(* CODESYS project WagoAppKNX.ecp

Project tree, tasks and I/O mapping:
  Steuerung : 750-8202 PFC200 2ETH RS, WAGO, order no. 0750-8202, version 5.14.3.31
    application Firmware_15
      libraries: ; WagoAppKNX, 1.0.2.6 (WAGO); VisuDialogs, * (System)
      task PLC_Task (cyclic, interval t#50ms, priority 15) calls PLC_PRG
      task VISU_TASK (cyclic, interval 100 ms, priority 15) calls VisuElems.Visu_Prg
      program PLC_PRG [CFC]
      visualisation Visualization
      Symbols
      program PLC_PRG_TP [CFC]
      visualisation Visualization_TM
    Kbus : Kbus, WAGO, version 1.4.0.2
        unmapped channels: K-BUS diagnostics
      KNX_EIB_TP1_Interface : 0753-0646, WAGO, order no. 0753-0646, version 0.0.0.10
          settings: K-BUS Module slot index = 1
          unmapped channels: _INPUTCHANNEL, _OUTPUTCHANNEL
    MODBUS
      MODBUS : MODBUS, WAGO, order no. n/a, version 1.1.1.15
    Serial
      COM1 : COM1, WAGO, version 0.0.0.19
  PFC200_2ETH_RS : 750-8202 PFC200 2ETH RS, WAGO, order no. 0750-8202, version 5.14.3.31
    application Application
      libraries: ; WagoAppKNX, 1.0.4.11 (WAGO)
      task PLC_Task (cyclic, interval t#50ms, priority 15) calls PLC_PRG
      program PLC_PRG [CFC]
    Kbus : Kbus, WAGO, version 1.4.0.2
        unmapped channels: K-BUS diagnostics
      _8_DI_Generic : 075x-8DI, WAGO, order no. 075x-8DI, version 0.0.0.13
          unmapped channels: _IN
      _2_DO_Generic : 075x-2DO, WAGO, order no. 075x-2DO, version 0.0.0.13
          unmapped channels: _OUT
      KNX_EIB_TP1_Interface : 0753-0646, WAGO, order no. 0753-0646, version 0.0.0.10
          unmapped channels: _INPUTCHANNEL, _OUTPUTCHANNEL
    MODBUS
      MODBUS : MODBUS, WAGO, order no. n/a, version 1.1.1.15
    Serial
      COM1 : COM1, WAGO, version 0.0.0.19
  PFC200_2ETH_RS_1 : 750-8202 PFC200 2ETH RS, WAGO, order no. 0750-8202, version 5.16.3.16
    application Firmware_19
      libraries: ; WagoAppKNX, 1.0.4.11 (WAGO); WagoSysKbusModule, 1.8.4.4 (WAGO); VisuDialogs, * (System)
      task PLC_Task (cyclic, interval t#50ms, priority 15) calls PLC_PRG
      task VISU_TASK (cyclic, interval 100 ms, priority 15) calls VisuElems.Visu_Prg
      program PLC_PRG [CFC]
      visualisation Visualization
      Symbols
    Kbus : Kbus, WAGO, version 1.4.0.2
        unmapped channels: K-BUS diagnostics
      KNX_EIB_TP1_Interface : 0753-0646, WAGO, order no. 0753-0646, version 0.0.0.10
          settings: K-BUS Module slot index = 1
          unmapped channels: _INPUTCHANNEL, _OUTPUTCHANNEL
    MODBUS
      MODBUS : MODBUS, WAGO, order no. n/a, version 1.1.1.16
    Serial
      COM1 : COM1, WAGO, version 0.0.0.19
  Firmware_11 : 750-8202 PFC200 2ETH RS, WAGO, order no. 0750-8202, version 5.11.1.16
    application Firmware_11
      libraries: ; WagoAppKNX, * (WAGO)
      task PLC_Task (cyclic, interval t#50ms, priority 15) calls PLC_PRG
      task VISU_TASK (cyclic, interval 100 ms, priority 15) calls VisuElems.Visu_Prg
      program PLC_PRG [CFC]
      Symbols
      visualisation Visualization
    Kbus : Kbus, WAGO, version 1.4.0.2
        unmapped channels: K-BUS diagnostics
      _16_DI_Generic : 075x-16DI, WAGO, order no. 075x-16DI, version 0.0.0.13
          settings: K-BUS Module slot index = 1
          unmapped channels: _IN
      _16_DI_Generic_1 : 075x-16DI, WAGO, order no. 075x-16DI, version 0.0.0.13
          settings: K-BUS Module slot index = 2
          unmapped channels: _IN
      _16_DI_Generic_2 : 075x-16DI, WAGO, order no. 075x-16DI, version 0.0.0.13
          settings: K-BUS Module slot index = 3
          unmapped channels: _IN
      _8_DI_Generic : 075x-8DI, WAGO, order no. 075x-8DI, version 0.0.0.13
          settings: K-BUS Module slot index = 4
          unmapped channels: _IN
      _8_DI_Generic_1 : 075x-8DI, WAGO, order no. 075x-8DI, version 0.0.0.13
          settings: K-BUS Module slot index = 5
          unmapped channels: _IN
      _16_DO_Generic : 075x-16DO, WAGO, order no. 075x-16DO, version 0.0.0.13
          settings: K-BUS Module slot index = 6
          unmapped channels: _OUT
      _16_DO_Generic_1 : 075x-16DO, WAGO, order no. 075x-16DO, version 0.0.0.13
          settings: K-BUS Module slot index = 7
          unmapped channels: _OUT
      _16_DO_Generic_2 : 075x-16DO, WAGO, order no. 075x-16DO, version 0.0.0.13
          settings: K-BUS Module slot index = 8
          unmapped channels: _OUT
      KNX_EIB_TP1_Interface : 0753-0646, WAGO, order no. 0753-0646, version 0.0.0.10
          settings: K-BUS Module slot index = 9
          unmapped channels: _INPUTCHANNEL, _OUTPUTCHANNEL
      DALI_MULTI_MASTER_MODULE : 0753-0647, WAGO, order no. 0753-0647, version 0.0.0.20
          settings: K-BUS Module slot index = 10
          unmapped channels: _IN, _OUT
    MODBUS
      MODBUS : MODBUS, WAGO, order no. n/a, version 1.1.1.15
    Serial
      COM1 : COM1, WAGO, version 0.0.0.19
  libraries: VisuSymbols, 4.1.0.0 (System); WagoVisuIcons, 1.1.0.5 (WAGO); WagoVisuIconsMaterialDesign, 1.0.0.0 (WAGO)
  text list GlobalTextList
*)

// Steuerung/Firmware_15/PLC_PRG
PROGRAM PLC_PRG
VAR
	KNX_Master: FbKNX_Master;
	oStatus: WagoAppKNX.WagoSysErrorBase.FbResult;
	sStatus: STRING;
	xProgMode: BOOL;
	wCountFbDPT: WORD;
	M1_001_DPT_Switch_Control: WagoAppKNX.FbDPT_Switch_Control;
	xUpdate_PLC: BOOL;
	xControl_OUT: BOOL;
	xSwitch_OUT: BOOL;
	dwIndex_DPT: DWORD := 1;
	xSwitch_IN: BOOL;
	xControl_IN: BOOL;
	xUpdate_KNX: BOOL;
END_VAR

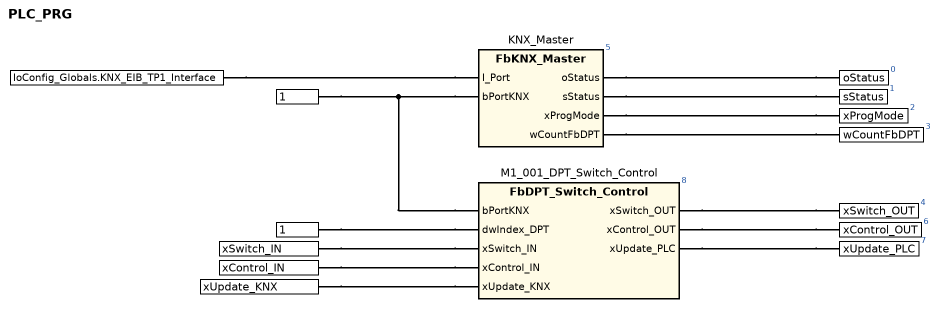
oStatus := KNX_Master.oStatus;
sStatus := KNX_Master.sStatus;
xProgMode := KNX_Master.xProgMode;
wCountFbDPT := KNX_Master.wCountFbDPT;
xSwitch_OUT := M1_001_DPT_Switch_Control.xSwitch_OUT;
KNX_Master(I_Port := IoConfig_Globals.KNX_EIB_TP1_Interface, bPortKNX := 1); // FbKNX_Master
xControl_OUT := M1_001_DPT_Switch_Control.xControl_OUT;
xUpdate_PLC := M1_001_DPT_Switch_Control.xUpdate_PLC;
M1_001_DPT_Switch_Control(
    bPortKNX := 1,
    dwIndex_DPT := 1,
    xSwitch_IN := xSwitch_IN,
    xControl_IN := xControl_IN,
    xUpdate_KNX := xUpdate_KNX); // FbDPT_Switch_Control

END_PROGRAM

// PFC200_2ETH_RS/Application/PLC_PRG
PROGRAM PLC_PRG
VAR
	KNX_Master: FbKNX_Master;
	oStatus: WagoAppKNX.WagoSysErrorBase.FbResult;
	sStatus: STRING;
	xProgMode: BOOL;
	wCountFbDPT: WORD;
	M1_001_DPT_Switch_Control: WagoAppKNX.FbDPT_Switch_Control;
	xUpdate_PLC: BOOL;
	xControl_OUT: BOOL;
	xSwitch_OUT: BOOL;
	dwIndex_DPT: DWORD := 1;
	xSwitch_IN: BOOL;
	xControl_IN: BOOL;
	xUpdate_KNX: BOOL;
END_VAR

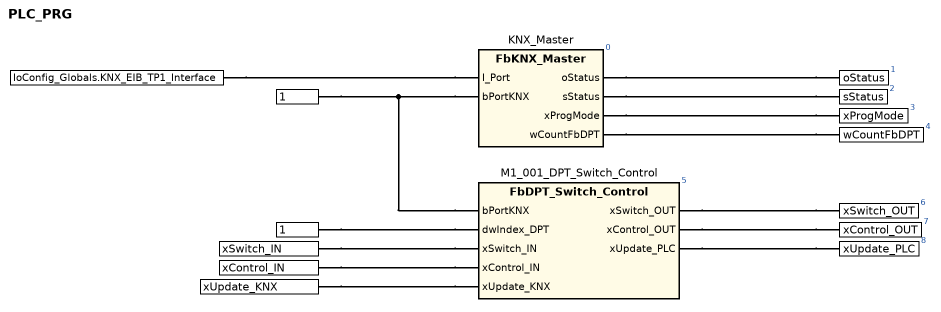
KNX_Master(I_Port := IoConfig_Globals.KNX_EIB_TP1_Interface, bPortKNX := 1); // FbKNX_Master
oStatus := KNX_Master.oStatus;
sStatus := KNX_Master.sStatus;
xProgMode := KNX_Master.xProgMode;
wCountFbDPT := KNX_Master.wCountFbDPT;
M1_001_DPT_Switch_Control(
    bPortKNX := 1,
    dwIndex_DPT := 1,
    xSwitch_IN := xSwitch_IN,
    xControl_IN := xControl_IN,
    xUpdate_KNX := xUpdate_KNX); // FbDPT_Switch_Control
xSwitch_OUT := M1_001_DPT_Switch_Control.xSwitch_OUT;
xControl_OUT := M1_001_DPT_Switch_Control.xControl_OUT;
xUpdate_PLC := M1_001_DPT_Switch_Control.xUpdate_PLC;

END_PROGRAM

// PFC200_2ETH_RS_1/Firmware_19/PLC_PRG
PROGRAM PLC_PRG
VAR
	KNX_Master: FbKNX_Master;
	oStatus: WagoAppKNX.WagoSysErrorBase.FbResult;
	sStatus: STRING;
	xProgMode: BOOL;
	wCountFbDPT: WORD;
	M1_001_DPT_Switch_Control: WagoAppKNX.FbDPT_Switch_Control;
	xUpdate_PLC: BOOL;
	xControl_OUT: BOOL;
	xSwitch_OUT: BOOL;
	dwIndex_DPT: DWORD := 1;
	xSwitch_IN: BOOL;
	xControl_IN: BOOL;
	xUpdate_KNX: BOOL;
END_VAR

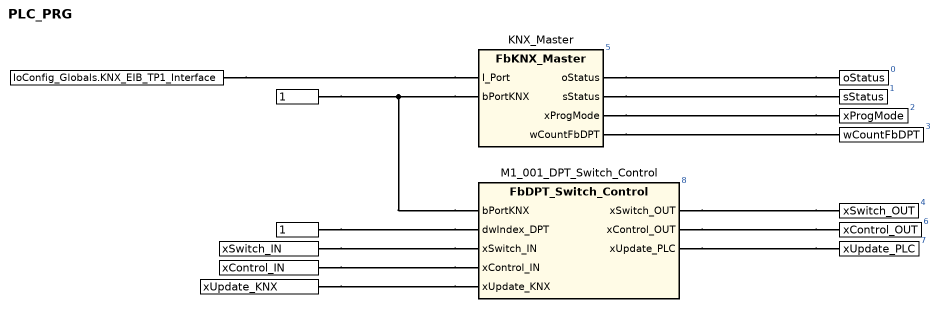
oStatus := KNX_Master.oStatus;
sStatus := KNX_Master.sStatus;
xProgMode := KNX_Master.xProgMode;
wCountFbDPT := KNX_Master.wCountFbDPT;
xSwitch_OUT := M1_001_DPT_Switch_Control.xSwitch_OUT;
KNX_Master(I_Port := IoConfig_Globals.KNX_EIB_TP1_Interface, bPortKNX := 1); // FbKNX_Master
xControl_OUT := M1_001_DPT_Switch_Control.xControl_OUT;
xUpdate_PLC := M1_001_DPT_Switch_Control.xUpdate_PLC;
M1_001_DPT_Switch_Control(
    bPortKNX := 1,
    dwIndex_DPT := 1,
    xSwitch_IN := xSwitch_IN,
    xControl_IN := xControl_IN,
    xUpdate_KNX := xUpdate_KNX); // FbDPT_Switch_Control

END_PROGRAM

// Firmware_11/Firmware_11/PLC_PRG
PROGRAM PLC_PRG
VAR
	KNX_Master: FbKNX_Master;
	oStatus: WagoAppKNX.WagoSysErrorBase.FbResult;
	sStatus: STRING;
	xProgMode: BOOL;
	wCountFbDPT: WORD;
	M1_001_DPT_Switch_Control: WagoAppKNX.FbDPT_Switch_Control;
	xUpdate_PLC: BOOL;
	xControl_OUT: BOOL;
	xSwitch_OUT: BOOL;
	dwIndex_DPT: DWORD := 1;
	xSwitch_IN: BOOL;
	xControl_IN: BOOL;
	xUpdate_KNX: BOOL;
END_VAR

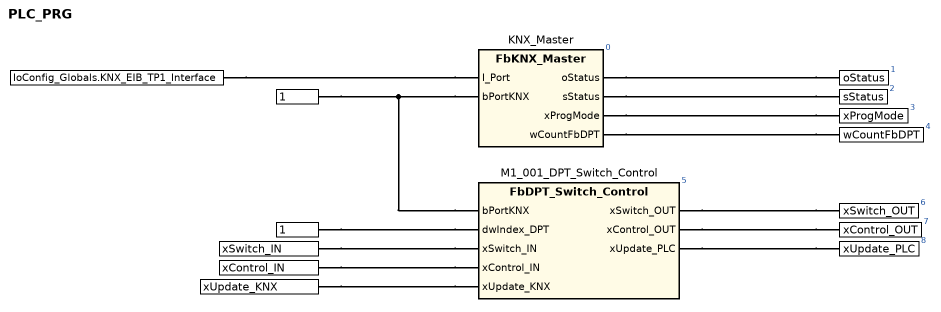
KNX_Master(I_Port := IoConfig_Globals.KNX_EIB_TP1_Interface, bPortKNX := 1); // FbKNX_Master
oStatus := KNX_Master.oStatus;
sStatus := KNX_Master.sStatus;
xProgMode := KNX_Master.xProgMode;
wCountFbDPT := KNX_Master.wCountFbDPT;
M1_001_DPT_Switch_Control(
    bPortKNX := 1,
    dwIndex_DPT := 1,
    xSwitch_IN := xSwitch_IN,
    xControl_IN := xControl_IN,
    xUpdate_KNX := xUpdate_KNX); // FbDPT_Switch_Control
xSwitch_OUT := M1_001_DPT_Switch_Control.xSwitch_OUT;
xControl_OUT := M1_001_DPT_Switch_Control.xControl_OUT;
xUpdate_PLC := M1_001_DPT_Switch_Control.xUpdate_PLC;

END_PROGRAM

// Steuerung/Firmware_15/PLC_PRG_TP
PROGRAM PLC_PRG_TP
VAR
	KNX_Master_TM: FbKNX_Master_TM;
	oStatus_TM: WagoAppKNX.WagoSysErrorBase.FbResult;
	sStatus_TM: STRING;
	stPhyAddress_TM: STRING(9) := '2.3.32';
	xFilter_Mode_TM: BOOL;
END_VAR

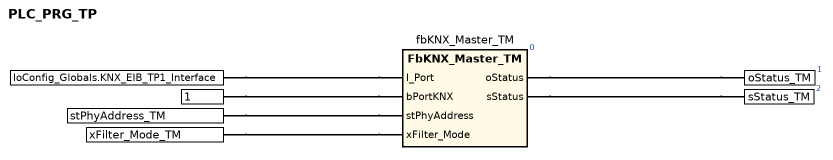
fbKNX_Master_TM(
    I_Port := IoConfig_Globals.KNX_EIB_TP1_Interface,
    bPortKNX := 1,
    stPhyAddress := stPhyAddress_TM,
    xFilter_Mode := xFilter_Mode_TM);
oStatus_TM := fbKNX_Master_TM.oStatus;
sStatus_TM := fbKNX_Master_TM.sStatus;

END_PROGRAM

// Steuerung/Firmware_15/Visualization
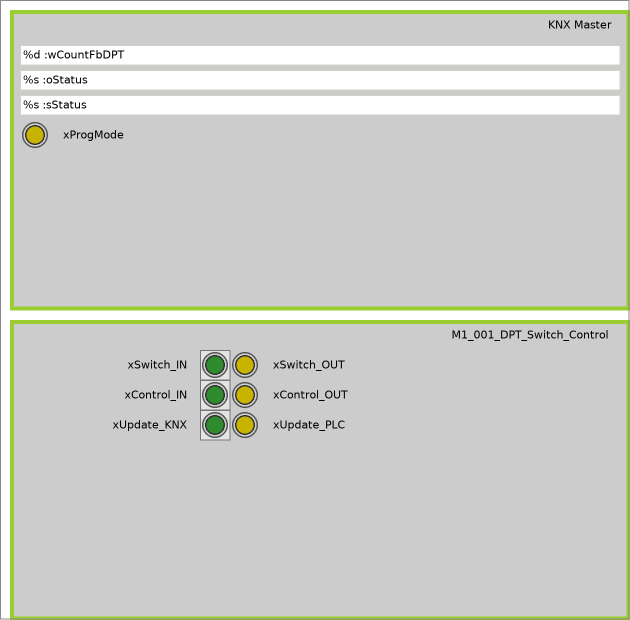
VISUALIZATION Visualization  // 630x620
    Rectangle (10,10 620x300)
    Label (530,10 100x30), "KNX Master"
    Textfield (20,70 600x20), "%s :oStatus", text variable: PLC_PRG.oStatus
        OnMouseClick: write the text variable via Default
    Textfield (20,95 600x20), "%s :sStatus", text variable: PLC_PRG.sStatus
        OnMouseClick: write the text variable via Default
    Lamp1 (20,120 30x30), variable: PLC_PRG.xProgMode, style: Lamp-Lamp1-Yellow
    Label (60,120 160x30), "xProgMode"
    Textfield (20,45 600x20), "%d :wCountFbDPT", text variable: PLC_PRG.wCountFbDPT
        OnMouseClick: write the text variable via Default
    Rectangle (10,320 620x300)
    Label (440,320 180x30), "M1_001_DPT_Switch_Control"
    PushSwitchLed (200,350 30x30), variable: PLC_PRG.xSwitch_IN, behaviour: TAP, style: Switch-PushSwitchLed-Green
    Label (90,350 100x30), "xSwitch_IN"
    PushSwitchLed (200,380 30x30), variable: PLC_PRG.xControl_IN, behaviour: TAP, style: Switch-PushSwitchLed-Green
    Label (90,380 100x30), "xControl_IN"
    Lamp1 (230,350 30x30), variable: PLC_PRG.xSwitch_OUT, style: Lamp-Lamp1-Yellow
    Label (270,350 160x30), "xSwitch_OUT"
    Lamp1 (230,380 30x30), variable: PLC_PRG.xControl_OUT, style: Lamp-Lamp1-Yellow
    Label (270,380 160x30), "xControl_OUT"
    PushSwitchLed (200,410 30x30), variable: PLC_PRG.xUpdate_KNX, behaviour: TAP, style: Switch-PushSwitchLed-Green
    Label (90,410 100x30), "xUpdate_KNX"
    Lamp1 (230,410 30x30), variable: PLC_PRG.xUpdate_PLC, style: Lamp-Lamp1-Yellow
    Label (270,410 160x30), "xUpdate_PLC"
END_VISUALIZATION

// Steuerung/Firmware_15/Visualization_TM
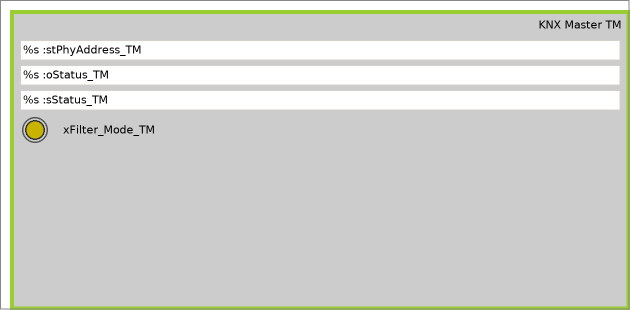
VISUALIZATION Visualization_TM  // 630x310
    Rectangle (10,10 620x300)
    Label (530,10 100x30), "KNX Master TM"
    Textfield (20,65 600x20), "%s :oStatus_TM", text variable: PLC_PRG.oStatus_TM
        OnMouseClick: write the text variable via Default
    Textfield (20,90 600x20), "%s :sStatus_TM", text variable: PLC_PRG.sStatus_TM
        OnMouseClick: write the text variable via Default
    Lamp1 (20,115 30x30), variable: PLC_PRG.xFilter_Mode_TM, style: Lamp-Lamp1-Yellow
    Label (60,115 160x30), "xFilter_Mode_TM"
    Textfield (20,40 600x20), "%s :stPhyAddress_TM", text variable: PLC_PRG.stPhyAddress_TM
        OnMouseClick: write the text variable via Default
END_VISUALIZATION

// PFC200_2ETH_RS_1/Firmware_19/Visualization
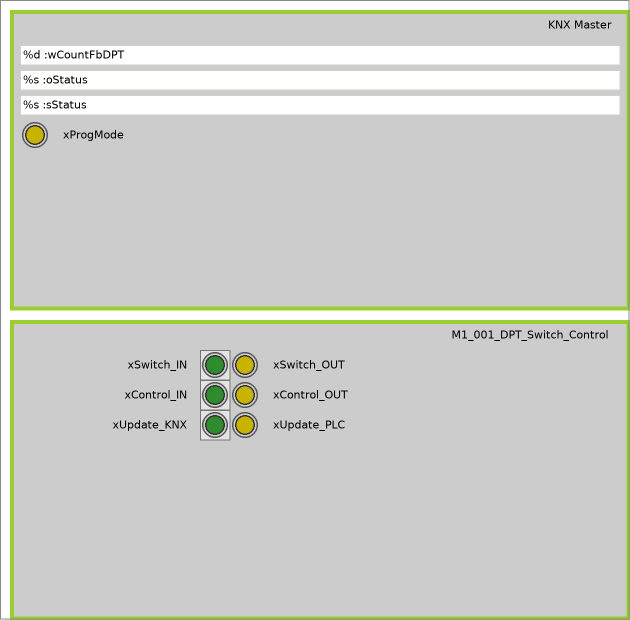
VISUALIZATION Visualization  // 630x620
    Rectangle (10,10 620x300)
    Label (530,10 100x30), "KNX Master"
    Textfield (20,70 600x20), "%s :oStatus", text variable: PLC_PRG.oStatus
        OnMouseClick: write the text variable via Default
    Textfield (20,95 600x20), "%s :sStatus", text variable: PLC_PRG.sStatus
        OnMouseClick: write the text variable via Default
    Lamp1 (20,120 30x30), variable: PLC_PRG.xProgMode, style: Lamp-Lamp1-Yellow
    Label (60,120 160x30), "xProgMode"
    Textfield (20,45 600x20), "%d :wCountFbDPT", text variable: PLC_PRG.wCountFbDPT
        OnMouseClick: write the text variable via Default
    Rectangle (10,320 620x300)
    Label (440,320 180x30), "M1_001_DPT_Switch_Control"
    PushSwitchLed (200,350 30x30), variable: PLC_PRG.xSwitch_IN, behaviour: TAP, style: Switch-PushSwitchLed-Green
    Label (90,350 100x30), "xSwitch_IN"
    PushSwitchLed (200,380 30x30), variable: PLC_PRG.xControl_IN, behaviour: TAP, style: Switch-PushSwitchLed-Green
    Label (90,380 100x30), "xControl_IN"
    Lamp1 (230,350 30x30), variable: PLC_PRG.xSwitch_OUT, style: Lamp-Lamp1-Yellow
    Label (270,350 160x30), "xSwitch_OUT"
    Lamp1 (230,380 30x30), variable: PLC_PRG.xControl_OUT, style: Lamp-Lamp1-Yellow
    Label (270,380 160x30), "xControl_OUT"
    PushSwitchLed (200,410 30x30), variable: PLC_PRG.xUpdate_KNX, behaviour: TAP, style: Switch-PushSwitchLed-Green
    Label (90,410 100x30), "xUpdate_KNX"
    Lamp1 (230,410 30x30), variable: PLC_PRG.xUpdate_PLC, style: Lamp-Lamp1-Yellow
    Label (270,410 160x30), "xUpdate_PLC"
END_VISUALIZATION

// Firmware_11/Firmware_11/Visualization
VISUALIZATION Visualization  // 2x2
END_VISUALIZATION
